// TIA Portal V19 export
DATA_BLOCK "Recv from AlcipM3"   // DB477
TITLE = Recv Interface from Flex A AlcipM3
{ S7_Optimized_Access := 'TRUE' }
// stored: AutoNumber false, MemoryReserve 0
   VAR RETAIN
      CC1 : Struct   // Alcip Comms Out - Cleaning Circuit 1 - Polygon Filler
         CL_CC_AckWdCnt : Int;
         CL_CC_CipOk2 : Bool;
         CL_CC_CipRun : Bool;
         CL_CC_CTHI : Bool;
         CL_CC_End : Bool;
         CL_CC_TTHI : Bool;
         CL_CC_Fault : Bool;
         CL_CC_CipReq : Bool;
         CL_CC_FilToTankExpired : Bool;
         CL_CC_spareByte : Byte;
         hmi : Struct
            commsFault : Bool;
            s1 : Bool;   // spare
            s2 : Bool;   // spare
            s3 : Bool;   // spare
            s4 : Bool;   // spare
            s5 : Bool;   // spare
            s6 : Bool;   // spare
            s7 : Bool;   // spare
            f1 : Bool;   // spare
            f2 : Bool;   // spare
            f3 : Bool;   // spare
            f4 : Bool;   // spare
            f5 : Bool;   // spare
            f6 : Bool;   // spare
            f7 : Bool;   // spare
            f8 : Bool;   // spare
         END_STRUCT;
      END_STRUCT;
      CC2 : Struct   // Alcip Comms Out - Cleaning Circuit 2 - FCL Filler
         CL_CC_AckWdCnt : Int;
         CL_CC_CipOk2 : Bool;
         CL_CC_CipRun : Bool;
         CL_CC_CTHI : Bool;
         CL_CC_End : Bool;
         CL_CC_TTHI : Bool;
         CL_CC_Fault : Bool;
         CL_CC_CipReq : Bool;
         CL_CC_FilToTankExpired : Bool;
         CL_CC_spareByte : Byte;
         dummySpace : Int;
      END_STRUCT;
      CC3 : Struct   // Alcip Comms Out - Cleaning Circuit 2 - Gasti Filler
         CL_CC_AckWdCnt : Int;
         CL_CC_CipOk2 : Bool;
         CL_CC_CipRun : Bool;
         CL_CC_CTHI : Bool;
         CL_CC_End : Bool;
         CL_CC_TTHI : Bool;
         CL_CC_Fault : Bool;
         CL_CC_CipReq : Bool;
         CL_CC_FilToTankExpired : Bool;
         CL_CC_spareByte : Byte;
         dummySpace : Int;
      END_STRUCT;
   END_VAR
BEGIN
END_DATA_BLOCK
